TYPE (* Typedef of the non-TP CAN Message *)
  (* Version 1.0, 2025-09-04, franz *)
  PACKAGE isobus;
  CAN_MSG : STRUCT
    data : ARRAY [0..7] OF BYTE := [16#FF, 16#FF, 16#FF, 16#FF, 16#FF, 16#FF, 16#FF, 16#FF];
  END_STRUCT;
END_TYPE
